SYSTEM Xquery
  (* Version 1.0, 2022-12-14, anubis *)
  APPLICATION selfInitializationApp
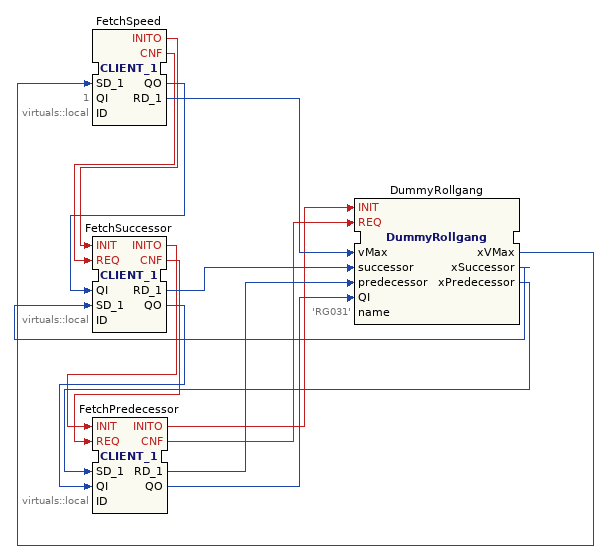
    FBS
      DummyRollgang : DummyRollgang(name := 'RG031');
      FetchSpeed : CLIENT_1(QI := 1, ID := virtuals::local);
      FetchSuccessor : CLIENT_1(ID := virtuals::local);
      FetchPredecessor : CLIENT_1(ID := virtuals::local);
    END_FBS
    EVENT_CONNECTIONS
      FetchSpeed.INITO TO FetchSuccessor.INIT;
      FetchSuccessor.INITO TO FetchPredecessor.INIT;
      FetchPredecessor.INITO TO DummyRollgang.INIT;
      FetchPredecessor.CNF TO DummyRollgang.REQ;
      FetchSpeed.CNF TO FetchSuccessor.REQ;
      FetchSuccessor.CNF TO FetchPredecessor.REQ;
    END_CONNECTIONS
    DATA_CONNECTIONS
      FetchSpeed.QO TO FetchSuccessor.QI;
      FetchSpeed.RD_1 TO DummyRollgang.vMax;
      FetchSuccessor.RD_1 TO DummyRollgang.successor;
      FetchPredecessor.RD_1 TO DummyRollgang.predecessor;
      FetchPredecessor.QO TO DummyRollgang.QI;
      DummyRollgang.xVMax TO FetchSpeed.SD_1;
      DummyRollgang.xSuccessor TO FetchSuccessor.SD_1;
      DummyRollgang.xPredecessor TO FetchPredecessor.SD_1;
      FetchSuccessor.QO TO FetchPredecessor.QI;
    END_CONNECTIONS
  END_APPLICATION
  DEVICE FORTE_PC : FORTE_PC(MGR_ID := "localhost:61499" (* Device manager socket ID *))
    {SET_ATTRIBUTE(Profile, HOLOBLOC)}
    RESOURCE Rollgang : EMB_RES
      EVENT_CONNECTIONS
        START.WARM TO selfInitializationApp.FetchSpeed.INIT;
        START.COLD TO selfInitializationApp.FetchSpeed.INIT;
      END_CONNECTIONS
    END_RESOURCE
  END_DEVICE
  MAPPINGS
    selfInitializationApp.DummyRollgang ON FORTE_PC.Rollgang;
    selfInitializationApp.FetchSpeed ON FORTE_PC.Rollgang;
    selfInitializationApp.FetchSuccessor ON FORTE_PC.Rollgang;
    selfInitializationApp.FetchPredecessor ON FORTE_PC.Rollgang;
  END_MAPPINGS
END_SYSTEM
